ABB RAPID module: RAPIDFile.mod

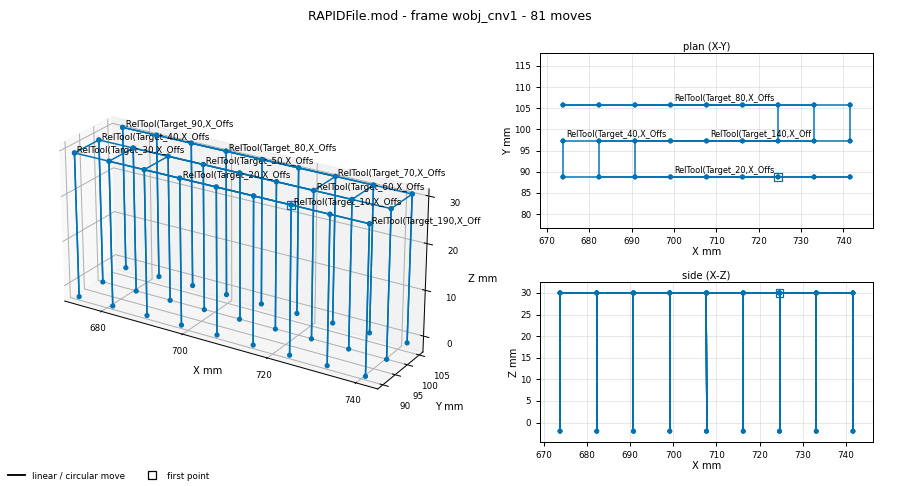
[picture p0: tool path of RAPIDFile.mod in frame wobj_cnv1, 81 of 81 moves have a stored position in this frame; points joined in program order, loops and branches not executed]
MODULE Module1
	PERS tooldata tPlungeDukane:=[TRUE,[[0,-0.14,318.999],[1,0,0,0]],[2.006,[0,-1.643,143.868],[1,0,0,0],0,0,0]];

   CONST robtarget Target_10:=[[703.4,110,0],[-1.5E-08,0.923879533,-0.382683432,3.5E-08],[0,0,0,0],[9E+09,9E+09,9E+09,9E+09,9E+09,0]];
   CONST robtarget Target_20:=[[678,110,0],[-1.5E-08,0.923879533,-0.382683432,3.5E-08],[0,0,0,0],[9E+09,9E+09,9E+09,9E+09,9E+09,0]];
   CONST robtarget Target_30:=[[652.6,110,0],[-1.5E-08,0.923879533,-0.382683432,3.5E-08],[0,0,0,0],[9E+09,9E+09,9E+09,9E+09,9E+09,0]];
   CONST robtarget Target_40:=[[652.6,118.5,0],[-1.5E-08,0.923879533,-0.382683432,3.5E-08],[0,0,0,0],[9E+09,9E+09,9E+09,9E+09,9E+09,0]];
   CONST robtarget Target_50:=[[678,118.5,0],[-1.5E-08,0.923879533,-0.382683432,3.5E-08],[0,0,0,0],[9E+09,9E+09,9E+09,9E+09,9E+09,0]];
   CONST robtarget Target_60:=[[703.4,118.5,0],[-1.5E-08,0.923879533,-0.382683432,3.5E-08],[0,0,0,0],[9E+09,9E+09,9E+09,9E+09,9E+09,0]];
   CONST robtarget Target_70:=[[703.4,127,0],[-1.5E-08,0.923879533,-0.382683432,3.5E-08],[0,0,0,0],[9E+09,9E+09,9E+09,9E+09,9E+09,0]];
   CONST robtarget Target_80:=[[678,127,0],[-1.5E-08,0.923879533,-0.382683432,3.5E-08],[0,0,0,0],[9E+09,9E+09,9E+09,9E+09,9E+09,0]];
   CONST robtarget Target_90:=[[652.6,127,0],[-1.5E-08,0.923879533,-0.382683432,3.5E-08],[0,0,0,0],[9E+09,9E+09,9E+09,9E+09,9E+09,0]];
   CONST robtarget Target_100:=[[661.1,127,0],[-1.5E-08,0.923879533,-0.382683432,3.5E-08],[0,0,0,0],[9E+09,9E+09,9E+09,9E+09,9E+09,0]];
   CONST robtarget Target_110:=[[686.5,127,0],[-1.5E-08,0.923879533,-0.382683432,3.5E-08],[0,0,0,0],[9E+09,9E+09,9E+09,9E+09,9E+09,0]];
   CONST robtarget Target_120:=[[711.9,127,0],[-1.5E-08,0.923879533,-0.382683432,3.5E-08],[0,0,0,0],[9E+09,9E+09,9E+09,9E+09,9E+09,0]];
   CONST robtarget Target_130:=[[711.9,118.5,0],[-1.5E-08,0.923879533,-0.382683432,3.5E-08],[0,0,0,0],[9E+09,9E+09,9E+09,9E+09,9E+09,0]];
   CONST robtarget Target_140:=[[686.5,118.5,0],[-1.5E-08,0.923879533,-0.382683432,3.5E-08],[0,0,0,0],[9E+09,9E+09,9E+09,9E+09,9E+09,0]];
   CONST robtarget Target_150:=[[661.1,118.5,0],[-1.5E-08,0.923879533,-0.382683432,3.5E-08],[0,0,0,0],[9E+09,9E+09,9E+09,9E+09,9E+09,0]];
   CONST robtarget Target_160:=[[661.1,110,0],[-1.5E-08,0.923879533,-0.382683432,3.5E-08],[0,0,0,0],[9E+09,9E+09,9E+09,9E+09,9E+09,0]];
   CONST robtarget Target_170:=[[686.5,110,0],[-1.5E-08,0.923879533,-0.382683432,3.5E-08],[0,0,0,0],[9E+09,9E+09,9E+09,9E+09,9E+09,0]];
   CONST robtarget Target_180:=[[711.9,110,0],[-1.5E-08,0.923879533,-0.382683432,3.5E-08],[0,0,0,0],[9E+09,9E+09,9E+09,9E+09,9E+09,0]];
   CONST robtarget Target_190:=[[720.4,110,0],[-1.5E-08,0.923879533,-0.382683432,3.5E-08],[0,0,0,0],[9E+09,9E+09,9E+09,9E+09,9E+09,0]];
   CONST robtarget Target_200:=[[695,110,0],[-1.5E-08,0.923879533,-0.382683432,3.5E-08],[0,0,0,0],[9E+09,9E+09,9E+09,9E+09,9E+09,0]];
   CONST robtarget Target_210:=[[669.6,110,0],[-1.5E-08,0.923879533,-0.382683432,3.5E-08],[0,0,0,0],[9E+09,9E+09,9E+09,9E+09,9E+09,0]];
   CONST robtarget Target_220:=[[669.6,118.5,0],[-1.5E-08,0.923879533,-0.382683432,3.5E-08],[0,0,0,0],[9E+09,9E+09,9E+09,9E+09,9E+09,0]];
   CONST robtarget Target_230:=[[695,118.5,0],[-1.5E-08,0.923879533,-0.382683432,3.5E-08],[0,0,0,0],[9E+09,9E+09,9E+09,9E+09,9E+09,0]];
   CONST robtarget Target_240:=[[720.4,118.5,0],[-1.5E-08,0.923879533,-0.382683432,3.5E-08],[0,0,0,0],[9E+09,9E+09,9E+09,9E+09,9E+09,0]];
   CONST robtarget Target_250:=[[720.4,127,0],[-1.5E-08,0.923879533,-0.382683432,3.5E-08],[0,0,0,0],[9E+09,9E+09,9E+09,9E+09,9E+09,0]];
   CONST robtarget Target_260:=[[695,127,0],[-1.5E-08,0.923879533,-0.382683432,3.5E-08],[0,0,0,0],[9E+09,9E+09,9E+09,9E+09,9E+09,0]];
   CONST robtarget Target_270:=[[669.6,127,0],[-1.5E-08,0.923879533,-0.382683432,3.5E-08],[0,0,0,0],[9E+09,9E+09,9E+09,9E+09,9E+09,0]];
   VAR num recipe := 2;    !1: r3295
                           !2: r7382
   VAR num X_Offset := 30;
   VAR num Y_Offset := 0;
   VAR num Z_CutDepth := -2;
   VAR num Z_ApproachHeight := -30;

   PROC main()
       ActUnit CNV1;
       ConfL \off;
       WHILE TRUE DO
           WaitWObj wobj_cnv1;

           Path_r3295;

       WaitRob \InPos;
       DropWObj wobj_cnv1;
       WaitTime 0.2;
       ENDWHILE
   ENDPROC

   PROC Path_r3295()
       MoveL RelTool(Target_10, X_Offset, Y_Offset, -30),v7000, z5, tPlungeDukane\WObj:= wobj_cnv1; MoveL RelTool(Target_10, X_Offset, Y_Offset, -Z_CutDepth),v7000,z1,tPlungeDukane\WObj:= wobj_cnv1; MoveL RelTool(Target_10, X_Offset, Y_Offset, -30),v7000, z5, tPlungeDukane\WObj:= wobj_cnv1;
       MoveL RelTool(Target_20, X_Offset, Y_Offset, -30),v7000, z5, tPlungeDukane\WObj:= wobj_cnv1; MoveL RelTool(Target_20, X_Offset, Y_Offset, -Z_CutDepth),v7000,z1,tPlungeDukane\WObj:= wobj_cnv1; MoveL RelTool(Target_20, X_Offset, Y_Offset, -30),v7000, z5, tPlungeDukane\WObj:= wobj_cnv1;
       MoveL RelTool(Target_30, X_Offset, Y_Offset, -30),v7000, z5, tPlungeDukane\WObj:= wobj_cnv1; MoveL RelTool(Target_30, X_Offset, Y_Offset, -Z_CutDepth),v7000,z1,tPlungeDukane\WObj:= wobj_cnv1; MoveL RelTool(Target_30, X_Offset, Y_Offset, -30),v7000, z5, tPlungeDukane\WObj:= wobj_cnv1;
       MoveL RelTool(Target_40, X_Offset, Y_Offset, -30),v7000, z5, tPlungeDukane\WObj:= wobj_cnv1; MoveL RelTool(Target_40, X_Offset, Y_Offset, -Z_CutDepth),v7000,z1,tPlungeDukane\WObj:= wobj_cnv1; MoveL RelTool(Target_40, X_Offset, Y_Offset, -30),v7000, z5, tPlungeDukane\WObj:= wobj_cnv1;
       MoveL RelTool(Target_50, X_Offset, Y_Offset, -30),v7000, z5, tPlungeDukane\WObj:= wobj_cnv1; MoveL RelTool(Target_50, X_Offset, Y_Offset, -Z_CutDepth),v7000,z1,tPlungeDukane\WObj:= wobj_cnv1; MoveL RelTool(Target_50, X_Offset, Y_Offset, -30),v7000, z5, tPlungeDukane\WObj:= wobj_cnv1;
       MoveL RelTool(Target_60, X_Offset, Y_Offset, -30),v7000, z5, tPlungeDukane\WObj:= wobj_cnv1; MoveL RelTool(Target_60, X_Offset, Y_Offset, -Z_CutDepth),v7000,z1,tPlungeDukane\WObj:= wobj_cnv1; MoveL RelTool(Target_60, X_Offset, Y_Offset, -30),v7000, z5, tPlungeDukane\WObj:= wobj_cnv1;
       MoveL RelTool(Target_70, X_Offset, Y_Offset, -30),v7000, z5, tPlungeDukane\WObj:= wobj_cnv1; MoveL RelTool(Target_70, X_Offset, Y_Offset, -Z_CutDepth),v7000,z1,tPlungeDukane\WObj:= wobj_cnv1; MoveL RelTool(Target_70, X_Offset, Y_Offset, -30),v7000, z5, tPlungeDukane\WObj:= wobj_cnv1;
       MoveL RelTool(Target_80, X_Offset, Y_Offset, -30),v7000, z5, tPlungeDukane\WObj:= wobj_cnv1; MoveL RelTool(Target_80, X_Offset, Y_Offset, -Z_CutDepth),v7000,z1,tPlungeDukane\WObj:= wobj_cnv1; MoveL RelTool(Target_80, X_Offset, Y_Offset, -30),v7000, z5, tPlungeDukane\WObj:= wobj_cnv1;
       MoveL RelTool(Target_90, X_Offset, Y_Offset, -30),v7000, z5, tPlungeDukane\WObj:= wobj_cnv1; MoveL RelTool(Target_90, X_Offset, Y_Offset, -Z_CutDepth),v7000,z1,tPlungeDukane\WObj:= wobj_cnv1; MoveL RelTool(Target_90, X_Offset, Y_Offset, -30),v7000, z5, tPlungeDukane\WObj:= wobj_cnv1;
       MoveL RelTool(Target_100, X_Offset, Y_Offset, -30),v7000, z5, tPlungeDukane\WObj:= wobj_cnv1; MoveL RelTool(Target_100, X_Offset, Y_Offset, -Z_CutDepth),v7000,z1,tPlungeDukane\WObj:= wobj_cnv1; MoveL RelTool(Target_100, X_Offset, Y_Offset, -30),v7000, z5, tPlungeDukane\WObj:= wobj_cnv1;
       MoveL RelTool(Target_110, X_Offset, Y_Offset, -30),v7000, z5, tPlungeDukane\WObj:= wobj_cnv1; MoveL RelTool(Target_110, X_Offset, Y_Offset, -Z_CutDepth),v7000,z1,tPlungeDukane\WObj:= wobj_cnv1; MoveL RelTool(Target_110, X_Offset, Y_Offset, -30),v7000, z5, tPlungeDukane\WObj:= wobj_cnv1;
       MoveL RelTool(Target_120, X_Offset, Y_Offset, -30),v7000, z5, tPlungeDukane\WObj:= wobj_cnv1; MoveL RelTool(Target_120, X_Offset, Y_Offset, -Z_CutDepth),v7000,z1,tPlungeDukane\WObj:= wobj_cnv1; MoveL RelTool(Target_120, X_Offset, Y_Offset, -30),v7000, z5, tPlungeDukane\WObj:= wobj_cnv1;
       MoveL RelTool(Target_130, X_Offset, Y_Offset, -30),v7000, z5, tPlungeDukane\WObj:= wobj_cnv1; MoveL RelTool(Target_130, X_Offset, Y_Offset, -Z_CutDepth),v7000,z1,tPlungeDukane\WObj:= wobj_cnv1; MoveL RelTool(Target_130, X_Offset, Y_Offset, -30),v7000, z5, tPlungeDukane\WObj:= wobj_cnv1;
       MoveL RelTool(Target_140, X_Offset, Y_Offset, -30),v7000, z5, tPlungeDukane\WObj:= wobj_cnv1; MoveL RelTool(Target_140, X_Offset, Y_Offset, -Z_CutDepth),v7000,z1,tPlungeDukane\WObj:= wobj_cnv1; MoveL RelTool(Target_140, X_Offset, Y_Offset, -30),v7000, z5, tPlungeDukane\WObj:= wobj_cnv1;
       MoveL RelTool(Target_150, X_Offset, Y_Offset, -30),v7000, z5, tPlungeDukane\WObj:= wobj_cnv1; MoveL RelTool(Target_150, X_Offset, Y_Offset, -Z_CutDepth),v7000,z1,tPlungeDukane\WObj:= wobj_cnv1; MoveL RelTool(Target_150, X_Offset, Y_Offset, -30),v7000, z5, tPlungeDukane\WObj:= wobj_cnv1;
       MoveL RelTool(Target_160, X_Offset, Y_Offset, -30),v7000, z5, tPlungeDukane\WObj:= wobj_cnv1; MoveL RelTool(Target_160, X_Offset, Y_Offset, -Z_CutDepth),v7000,z1,tPlungeDukane\WObj:= wobj_cnv1; MoveL RelTool(Target_160, X_Offset, Y_Offset, -30),v7000, z5, tPlungeDukane\WObj:= wobj_cnv1;
       MoveL RelTool(Target_170, X_Offset, Y_Offset, -30),v7000, z5, tPlungeDukane\WObj:= wobj_cnv1; MoveL RelTool(Target_170, X_Offset, Y_Offset, -Z_CutDepth),v7000,z1,tPlungeDukane\WObj:= wobj_cnv1; MoveL RelTool(Target_170, X_Offset, Y_Offset, -30),v7000, z5, tPlungeDukane\WObj:= wobj_cnv1;
       MoveL RelTool(Target_180, X_Offset, Y_Offset, -30),v7000, z5, tPlungeDukane\WObj:= wobj_cnv1; MoveL RelTool(Target_180, X_Offset, Y_Offset, -Z_CutDepth),v7000,z1,tPlungeDukane\WObj:= wobj_cnv1; MoveL RelTool(Target_180, X_Offset, Y_Offset, -30),v7000, z5, tPlungeDukane\WObj:= wobj_cnv1;
       MoveL RelTool(Target_190, X_Offset, Y_Offset, -30),v7000, z5, tPlungeDukane\WObj:= wobj_cnv1; MoveL RelTool(Target_190, X_Offset, Y_Offset, -Z_CutDepth),v7000,z1,tPlungeDukane\WObj:= wobj_cnv1; MoveL RelTool(Target_190, X_Offset, Y_Offset, -30),v7000, z5, tPlungeDukane\WObj:= wobj_cnv1;
       MoveL RelTool(Target_200, X_Offset, Y_Offset, -30),v7000, z5, tPlungeDukane\WObj:= wobj_cnv1; MoveL RelTool(Target_200, X_Offset, Y_Offset, -Z_CutDepth),v7000,z1,tPlungeDukane\WObj:= wobj_cnv1; MoveL RelTool(Target_200, X_Offset, Y_Offset, -30),v7000, z5, tPlungeDukane\WObj:= wobj_cnv1;
       MoveL RelTool(Target_210, X_Offset, Y_Offset, -30),v7000, z5, tPlungeDukane\WObj:= wobj_cnv1; MoveL RelTool(Target_210, X_Offset, Y_Offset, -Z_CutDepth),v7000,z1,tPlungeDukane\WObj:= wobj_cnv1; MoveL RelTool(Target_210, X_Offset, Y_Offset, -30),v7000, z5, tPlungeDukane\WObj:= wobj_cnv1;
       MoveL RelTool(Target_220, X_Offset, Y_Offset, -30),v7000, z5, tPlungeDukane\WObj:= wobj_cnv1; MoveL RelTool(Target_220, X_Offset, Y_Offset, -Z_CutDepth),v7000,z1,tPlungeDukane\WObj:= wobj_cnv1; MoveL RelTool(Target_220, X_Offset, Y_Offset, -30),v7000, z5, tPlungeDukane\WObj:= wobj_cnv1;
       MoveL RelTool(Target_230, X_Offset, Y_Offset, -30),v7000, z5, tPlungeDukane\WObj:= wobj_cnv1; MoveL RelTool(Target_230, X_Offset, Y_Offset, -Z_CutDepth),v7000,z1,tPlungeDukane\WObj:= wobj_cnv1; MoveL RelTool(Target_230, X_Offset, Y_Offset, -30),v7000, z5, tPlungeDukane\WObj:= wobj_cnv1;
       MoveL RelTool(Target_240, X_Offset, Y_Offset, -30),v7000, z5, tPlungeDukane\WObj:= wobj_cnv1; MoveL RelTool(Target_240, X_Offset, Y_Offset, -Z_CutDepth),v7000,z1,tPlungeDukane\WObj:= wobj_cnv1; MoveL RelTool(Target_240, X_Offset, Y_Offset, -30),v7000, z5, tPlungeDukane\WObj:= wobj_cnv1;
       MoveL RelTool(Target_250, X_Offset, Y_Offset, -30),v7000, z5, tPlungeDukane\WObj:= wobj_cnv1; MoveL RelTool(Target_250, X_Offset, Y_Offset, -Z_CutDepth),v7000,z1,tPlungeDukane\WObj:= wobj_cnv1; MoveL RelTool(Target_250, X_Offset, Y_Offset, -30),v7000, z5, tPlungeDukane\WObj:= wobj_cnv1;
       MoveL RelTool(Target_260, X_Offset, Y_Offset, -30),v7000, z5, tPlungeDukane\WObj:= wobj_cnv1; MoveL RelTool(Target_260, X_Offset, Y_Offset, -Z_CutDepth),v7000,z1,tPlungeDukane\WObj:= wobj_cnv1; MoveL RelTool(Target_260, X_Offset, Y_Offset, -30),v7000, z5, tPlungeDukane\WObj:= wobj_cnv1;
       MoveL RelTool(Target_270, X_Offset, Y_Offset, -30),v7000, z5, tPlungeDukane\WObj:= wobj_cnv1; MoveL RelTool(Target_270, X_Offset, Y_Offset, -Z_CutDepth),v7000,z1,tPlungeDukane\WObj:= wobj_cnv1; MoveL RelTool(Target_270, X_Offset, Y_Offset, -30),v7000, z5, tPlungeDukane\WObj:= wobj_cnv1;
   ENDPROC
ENDMODULE
